{attribute 'GeneratedUsingTerminal: EK1501-0000-0016'}
{attribute addProperty BoxType "EK1501-0000-0016"}
{attribute addProperty Description "EK1501 EtherCAT Coupler (2A E-Bus, FX-MultiMode, ID switch)"}
{attribute addProperty Physics "YKY"}
{attribute addProperty Id "IDAT %I*ID_07C9D28F2WcStateAT %I*WcState_9091E0EB2InfoDataAT %I*InfoData_6F19DB2B2"}
{attribute addProperty CRC "2508032143"}
{attribute addProperty Size "6"}
TYPE EK1501_957D888F EXTENDS EtcSlaveBoxBase_77A0E4A7 :
STRUCT
	{attribute addProperty Name "ID"}
	ID : ID_07C9D28F;
	{attribute addProperty Name "WcState"}
	WcState : WcState_9091E0EB;
	{attribute addProperty Name "InfoData"}
	InfoData : InfoData_6F19DB2B;
END_STRUCT
END_TYPE

(* stored: Version 1.2.0.0, ProductVersion 3.1.4024.9
   DUT EK1501_957D888F: Id {2230bf8b-cb6a-4ee1-8681-a9d906f496f7} *)
